// TwinCAT 3 PLC project Untitled1
// ProgramVersion: 3.1.4024.0
// libraries:
//   Tc2_MC2, * (Beckhoff Automation GmbH)
//   Tc2_SerialCom, * (Beckhoff Automation GmbH)
//   Tc2_Standard, * (Beckhoff Automation GmbH)
//   Tc2_System, * (Beckhoff Automation GmbH)
//   Tc3_Module, * (Beckhoff Automation GmbH)
// project tree:
//   DUTs/ tDataFrame.TcDUT
//   GVLs/ GVL.TcGVL
//   / PlcTask.TcTTO, RS485task.TcTTO
//   POUs/ FB_Azimuth.TcPOU, FB_Elevation.TcPOU, FB_485.TcPOU, FB_Trinamic_motors.TcPOU, MAIN.TcPOU, RS485_prg.TcPOU
// real-time tasks:
//   TASK PlcTask: cycle T#10ms, priority 20, ADS port 350
//   TASK RS485task: cycle T#1ms, priority 21, ADS port 352
// motion (NC):
//   TASK NC-Task 1 SAF: cycle T#2ms, priority 4, ADS port 501
//   TASK NC-Task 1 SVB: cycle T#10ms, priority 8, ADS port 511
//   AXIS Axis 3 (id 3)
//     General: UnitName=°
//     Dynamic: Acceleration=15000, Deceleration=15000, Jerk=64125
//     Velo: RefSearch=142.5, RefSync=142.5, SlowManual=712.5, FastManual=4275, Fast=14250, Maximum=14250
//     PositionAreaControl: Enable=false
//     TargetPosControl: Enable=false
//     OtherSettings: AllowMotionCmdToSlave=true
//     encoder EncType=8
//       EncPara: ScaleFactorNumerator=360, ScaleFactorDenominator=1048576, MaxCount=#xffffffff, EncPositionSource=1
//     drive DrvType=9
//       DrvPara: MaxCount=#xffffffff, DriveControlDWord=#x00030100
//         Analog: VeloReferenz=15675, VeloScale=1.02400649589962, TorqueSetpointScale=10, ScaleFactorActTorque=0.1
//         TimeComp: TaskDelayCycles=1
//     controller CtrType=1
//       CtrPara: PriorControlFactor=1
//         PosDiffControl: Enable=false
//         Observer: BandWidth=20
// I/O:
//   DEVICE Device 1 (EtherCAT), AmsNetId 5.79.241.154.2.1
//     Term 1 (EK1200) [EK1200-5000 EtherCAT Power supply (2A E-Bus)]
//       Term 2 (EL7342) [EL7342 2Ch. DC motor output stage (50V, 3.5A)]
//       RS485_term [EL6021 Interface (RS422/485)]
//       Term 3 (EK1110) [EK1110 EtherCAT extension]
//     Drive 4 (AX5203-0000-0214) [AX5203-0000-0214 EtherCAT Drive (SoE, 2 Ch.)]
// variable links:
//   NC-Task 1 SAF/Axes/Axis 3 <-> Device 1 (EtherCAT)/Drive 4 (AX5203-0000-0214)
//     Drive/Inputs/In/nDataIn1 <-> AT 1/Following distance
//     Drive/Inputs/In/nDataIn3[0] <-> AT 1/Torque/force feedback value
//     Drive/Inputs/In/nDcOutputTime <-> InfoData/DcOutputShift
//     Drive/Inputs/In/nState1 <-> AT 1/Drive status word @bit 8
//     Drive/Inputs/In/nState2 <-> AT 1/Drive status word
//     Drive/Inputs/In/nState4 @bit 1 <-> WcState/InputToggle
//     Drive/Inputs/In/nState4 <-> WcState/WcState
//     Drive/Outputs/Out/nCtrl1 <-> MDT 1/Master control word @bit 8
//     Drive/Outputs/Out/nDataOut1 <-> MDT 1/Position command value
//     Enc/Inputs/In/nDataIn1 <-> AT 1/Position feedback 1 value
//     Enc/Inputs/In/nDcInputTime <-> InfoData/DcInputShift
//     Enc/Inputs/In/nState4 @bit 1 <-> WcState/InputToggle
//     Enc/Inputs/In/nState4 <-> WcState/WcState
//   Untitled1/Untitled1 Instance <-> Device 1 (EtherCAT)/Term 1 (EK1200)/Term 2 (EL7342)
//     PlcTask Inputs/MAIN.Elevation.Encoder_Value <-> ENC Status Channel 1/Counter value
//     PlcTask Inputs/MAIN.Elevation.Error <-> DCM Status Channel 1/Status/Error
//     PlcTask Inputs/MAIN.Elevation.Homing_Switch <-> DCM Status Channel 1/Status/Digital input 1
//     PlcTask Inputs/MAIN.Elevation.Limit_Switch <-> DCM Status Channel 1/Status/Digital input 2
//     PlcTask Inputs/MAIN.Elevation.Moving_negative <-> DCM Status Channel 1/Status/Moving negative
//     PlcTask Inputs/MAIN.Elevation.Moving_positive <-> DCM Status Channel 1/Status/Moving positive
//     PlcTask Inputs/MAIN.Elevation.Ready <-> DCM Status Channel 1/Status/Ready
//     PlcTask Inputs/MAIN.Elevation.Warning <-> DCM Status Channel 1/Status/Warning
//     PlcTask Outputs/MAIN.Elevation.Enable <-> DCM Control Channel 1/Control/Enable
//     PlcTask Outputs/MAIN.Elevation.Encoder_Setvalue <-> ENC Control Channel 1/Set counter value
//     PlcTask Outputs/MAIN.Elevation.Reset <-> DCM Control Channel 1/Control/Reset
//     PlcTask Outputs/MAIN.Elevation.Set_Encoder <-> ENC Control Channel 1/Control/Set counter
//     PlcTask Outputs/MAIN.Elevation.Target_Position <-> DCM Position Channel 1/Position
//   Untitled1/Untitled1 Instance <-> NC-Task 1 SAF/Axes/Axis 3
//     PlcTask Inputs/MAIN.Azimuth.Azimuth_axis.NcToPlc <-> Outputs/ToPlc
//     PlcTask Outputs/MAIN.Azimuth.Azimuth_axis.PlcToNc <-> Inputs/FromPlc

CONFIGURATION Untitled1
    RESOURCE PLC ON TwinCAT3
        TASK PlcTask(INTERVAL := T#10ms, PRIORITY := 20);
        TASK RS485task(INTERVAL := T#1ms, PRIORITY := 21);
        PROGRAM MAIN WITH PlcTask : MAIN;
        PROGRAM RS485_prg WITH RS485task : RS485_prg;
    END_RESOURCE
END_CONFIGURATION

// ---- DUTs/tDataFrame.TcDUT
TYPE tDataFrame : ARRAY[0..8] OF BYTE; END_TYPE

// ---- GVLs/GVL.TcGVL
{attribute 'qualified_only'}
VAR_GLOBAL


nSetBaudrate : DINT := 38400;	
	
	
		{attribute 'TcLinkTo' := '
								.D[0]   := TIIB[RS485_term]^COM TxPDO-Map Inputs^Data In 0;
                              	.D[1]   := TIIB[RS485_term]^COM TxPDO-Map Inputs^Data In 1;
								.D[2]   := TIIB[RS485_term]^COM TxPDO-Map Inputs^Data In 2;
								.D[3]   := TIIB[RS485_term]^COM TxPDO-Map Inputs^Data In 3;
								.D[4]   := TIIB[RS485_term]^COM TxPDO-Map Inputs^Data In 4;
								.D[5]   := TIIB[RS485_term]^COM TxPDO-Map Inputs^Data In 5;
								.D[6]   := TIIB[RS485_term]^COM TxPDO-Map Inputs^Data In 6;
								.D[7]   := TIIB[RS485_term]^COM TxPDO-Map Inputs^Data In 7;
								.D[8]   := TIIB[RS485_term]^COM TxPDO-Map Inputs^Data In 8;
								.D[9]   := TIIB[RS485_term]^COM TxPDO-Map Inputs^Data In 9;
								.D[10]  := TIIB[RS485_term]^COM TxPDO-Map Inputs^Data In 10;
								.D[11]  := TIIB[RS485_term]^COM TxPDO-Map Inputs^Data In 11;
								.D[12]  := TIIB[RS485_term]^COM TxPDO-Map Inputs^Data In 12;
								.D[13]  := TIIB[RS485_term]^COM TxPDO-Map Inputs^Data In 13;
								.D[14]  := TIIB[RS485_term]^COM TxPDO-Map Inputs^Data In 14;
								.D[15]  := TIIB[RS485_term]^COM TxPDO-Map Inputs^Data In 15;
								.D[16]  := TIIB[RS485_term]^COM TxPDO-Map Inputs^Data In 16;
								.D[17]  := TIIB[RS485_term]^COM TxPDO-Map Inputs^Data In 17;
								.D[18]  := TIIB[RS485_term]^COM TxPDO-Map Inputs^Data In 18;
								.D[19]  := TIIB[RS485_term]^COM TxPDO-Map Inputs^Data In 19;
								.D[20]  := TIIB[RS485_term]^COM TxPDO-Map Inputs^Data In 20;
								.D[21]  := TIIB[RS485_term]^COM TxPDO-Map Inputs^Data In 21;
								.Status := TIIB[RS485_term]^COM TxPDO-Map Inputs^Status'}							  
	COMin_EL6021_MASTER AT %I* : EL6inData22B;              

			{attribute 'TcLinkTo' := '
								.D[0]   := TIIB[RS485_term]^COM RxPDO-Map Outputs^Data Out 0;
                              	.D[1]   := TIIB[RS485_term]^COM RxPDO-Map Outputs^Data Out 1;
								.D[2]   := TIIB[RS485_term]^COM RxPDO-Map Outputs^Data Out 2;
								.D[3]   := TIIB[RS485_term]^COM RxPDO-Map Outputs^Data Out 3;
								.D[4]   := TIIB[RS485_term]^COM RxPDO-Map Outputs^Data Out 4;
								.D[5]   := TIIB[RS485_term]^COM RxPDO-Map Outputs^Data Out 5;
								.D[6]   := TIIB[RS485_term]^COM RxPDO-Map Outputs^Data Out 6;
								.D[7]   := TIIB[RS485_term]^COM RxPDO-Map Outputs^Data Out 7;
								.D[8]   := TIIB[RS485_term]^COM RxPDO-Map Outputs^Data Out 8;
								.D[9]   := TIIB[RS485_term]^COM RxPDO-Map Outputs^Data Out 9;
								.D[10]  := TIIB[RS485_term]^COM RxPDO-Map Outputs^Data Out 10;
								.D[11]  := TIIB[RS485_term]^COM RxPDO-Map Outputs^Data Out 11;
								.D[12]  := TIIB[RS485_term]^COM RxPDO-Map Outputs^Data Out 12;
								.D[13]  := TIIB[RS485_term]^COM RxPDO-Map Outputs^Data Out 13;
								.D[14]  := TIIB[RS485_term]^COM RxPDO-Map Outputs^Data Out 14;
								.D[15]  := TIIB[RS485_term]^COM RxPDO-Map Outputs^Data Out 15;
								.D[16]  := TIIB[RS485_term]^COM RxPDO-Map Outputs^Data Out 16;
								.D[17]  := TIIB[RS485_term]^COM RxPDO-Map Outputs^Data Out 17;
								.D[18]  := TIIB[RS485_term]^COM RxPDO-Map Outputs^Data Out 18;
								.D[19]  := TIIB[RS485_term]^COM RxPDO-Map Outputs^Data Out 19;
								.D[20]  := TIIB[RS485_term]^COM RxPDO-Map Outputs^Data Out 20;
								.D[21]  := TIIB[RS485_term]^COM RxPDO-Map Outputs^Data Out 21;
								.Ctrl   := TIIB[RS485_term]^COM RxPDO-Map Outputs^Ctrl'}	
	COMout_EL6021_MASTER AT %Q* : EL6outData22B;
	RxBuffer_MASTER : Combuffer;
	TxBuffer_MASTER : Combuffer;	

END_VAR

// ---- POUs/MAIN.TcPOU
PROGRAM MAIN
VAR
Elevation : FB_Elevation;
Azimuth : FB_Azimuth;
END_VAR

Elevation();
Azimuth();

END_PROGRAM

// ---- POUs/FB_Elevation.TcPOU
FUNCTION_BLOCK FB_Elevation
VAR_INPUT
END_VAR
VAR_OUTPUT
END_VAR
VAR
	
	//Data for ADS communtication
	Targetpos_mm 			: LREAL	:= 0;		//Data FROM ADS
	Targetpos_deg			: LREAL := 0;		//Data FROM ADS
	Current_Position_mm 	: LREAL;			//Data TO ADS
	Current_Position_deg 	: LREAL; 			//Data from inclonometer, updated asynchronous from RS485
	Enable AT %Q* 			: BOOL 	:= FALSE;	//Data FROM ADS
	Homeing 				: BOOL 	:= FALSE;	//Data TO ADS
	Homeing_Error 			: BOOL 	:= FALSE;	//Data TO ADS
	Homeing_Wrong_direction : BOOL  := FALSE;	//Data TO ADS
	Reset_requested 		: BOOL  := FALSE;	//Data FROM ADS
	Error AT %I* 			: BOOL;				//Data TO ADS
	Target_in_deg			: BOOL  := FALSE;	//DATA FROM ADS
	//Position_Error AT %I* 	: BOOL;
	
		
	//Data for ADS communtication END
	
	
	Reset AT %Q* 			: BOOL 	:= FALSE;
	Encoder_Value AT %I* : UDINT;
	Homing_Switch AT %I* : BOOL;
	Limit_Switch AT %I* : BOOL;
	Warning AT %I* : BOOL;

	Ready AT %I* : BOOL;
	Moving_positive AT %I* : BOOL;
	Moving_negative AT %I* : BOOL;
	//In_target AT %I* : BOOL;
	Set_Encoder AT %Q* : BOOL;
	Encoder_Setvalue AT %Q* : UDINT;
	Target_Position AT %Q* : UDINT;
	
	P_error : LREAL; //position error
	Ang_P_fac : REAL := 0.01; //This is not really a P factor, I think it's more of a I
 	//Ang_I_fac : REAL := 0.001;

	
	//firstrun :BOOL := TRUE;
	Homed : BOOL := FALSE;
	Homeing_Allowed : BOOL := TRUE;
	Homeing_State : UINT := 0;
	Reset_state : UINT := 0;
	
	Homing_started_mm : LREAL; // to monitor if the homeing goes the right direction
	
	Homeing_Timer : TON; //used for timeouts
	Homeing_Timer2 : TON;
END_VAR

VAR CONSTANT
	maxmove_mm : LREAL := 210;
	minmove_mm : LREAL := 0;
	Zeroposition : UDINT := 1000000;
END_VAR

IF Homeing_Error THEN
	enable := FALSE;
	Homeing_state := 0;
	Homed := FALSE;
END_IF

IF Reset_requested THEN
	Reset_Elevation();
END_IF

IF Homed = FALSE AND Enable = TRUE AND Homeing_Allowed AND Homeing_Error = FALSE THEN
	//The homing sequence should start automaticly if the PLC is restarted and Enable is set
	Homeing_sequence();
ELSE
	IF Homed = TRUE AND Enable = TRUE THEN //Normal operation
		IF Target_in_deg = FALSE THEN
			//'Dumb' positioning, semi-openloop the position is only based on the 
			//Encoder value, not the actual measured value
			Target_Position := mm_to_encoder(LIMIT(minmove_mm,targetpos_mm,maxmove_mm));
		ELSE
			//closed-loop positionin with a inclonometer in the loop
			P_error := Current_Position_deg - Targetpos_deg;
			Target_Position := mm_to_encoder(LIMIT(minmove_mm,
			Target_Position + P_error*Ang_P_fac
			,maxmove_mm));
		END_IF
	
	
		
	END_IF
END_IF

current_position_mm := encoder_to_mm(Encoder_Value);

METHOD encoder_to_mm : LREAL
VAR_INPUT
	encoder_pos : UDINT;
END_VAR

VAR
	encoder_ppr : LREAL := 2000;
	mm_per_rev : LREAL := 0.8; //calibrate this value
END_VAR
encoder_to_mm := UDINT_TO_LREAL(encoder_pos - Zeroposition) / (encoder_ppr * mm_per_rev);
END_METHOD

METHOD Homeing_sequence : BOOL
VAR_INPUT
END_VAR
VAR
	diff_pos : LREAL;
END_VAR
Homeing_Timer(IN:=TRUE, PT:= T#200S); //timeout of the homeing, it takes a long time to home...
Homeing := TRUE;

IF Homeing_Timer.Q THEN
	//Timeout as been reached
	Homeing_Error := TRUE;
	Homeing_Timer(IN:=FALSE);

END_IF

IF Homing_Switch AND Homeing_state < 3 THEN
	Homeing_state := 3;
END_IF

CASE Homeing_state OF
	0:
	 	//We want to set the current position to a high number so we can go into the negative as the countervalue is a UDINT
		Encoder_Setvalue := Zeroposition;
		Target_Position  := Zeroposition;
		Set_Encoder := 1;
		Homeing_Timer2(IN:= TRUE, PT:= T#1S);
		IF Homeing_Timer2.Q THEN
			Homeing_Timer2(IN:=FALSE);
			Homeing_state := 1;
		END_IF
			
	1:
		Set_Encoder := 0;
		
		Homeing_Timer2(IN:= TRUE, PT:= T#1S);
		IF Homeing_Timer2.Q THEN
			Homeing_Timer2(IN:=FALSE);
			Homeing_state := 2;
			Homing_started_mm := encoder_to_mm(Encoder_Value);
		END_IF
	2: 
		//Goes to a position in the 'negatives' 
		Target_Position := 0;
		diff_pos := (encoder_to_mm(Encoder_Value) - Homing_started_mm);
		//Diff_pos will be very large if it is going the correct direction due to underflow
		//If it does not grow large, it is going the wrong way 
		IF  diff_pos > 1 AND diff_pos < 1000 THEN
			// for some reason this happens sometime
			homeing_error := TRUE;
			Homeing_Wrong_direction := TRUE;
		END_IF
		
	3: 
		//Stop the motor and set the new zero when the motor has stopped
		Target_Position := Encoder_Value; //Stop the motor without disabling it
		Homeing_Timer2(IN:= TRUE, PT:= T#2S);
		IF Homeing_Timer2.Q THEN
			Encoder_Setvalue := Zeroposition;
			Target_Position := Zeroposition;
			Set_Encoder := 1;
			Homeing_state := 4;
			Homeing_Timer2(IN:=FALSE);
		END_IF
		
	4: 
	
		//Motor has been homed
		Set_Encoder := 0;
		Homeing_Timer(IN:=FALSE);
		Homeing := FALSE;
		Homed := TRUE;
		homeing_state := 0;
		
	
END_CASE
END_METHOD

METHOD mm_to_encoder : UDINT
VAR_INPUT
	mm_in : LREAL;
END_VAR
VAR
	encoder_ppr : LREAL := 2000;
	mm_per_rev : LREAL := 0.8; //calibrate this value
END_VAR
mm_to_encoder := LREAL_TO_UDINT(mm_in* mm_per_rev * encoder_ppr) + Zeroposition;
END_METHOD

METHOD Reset_Elevation : BOOL
VAR_INPUT
END_VAR

CASE Reset_state OF
	0:
		enable := FALSE;
		Reset_state := 1;
	1:
		Reset := TRUE;
		Targetpos_mm := Current_Position_mm ;
		Homed := FALSE;
		Homeing_Error := FALSE;
		Homeing_Wrong_direction := FALSE;
		Homeing_State := 0;
		Reset_state := 2;
		
	2: 
		Reset := FALSE;
		Reset_state := 3;
		
	3: //A extra one for good luck
		Reset := TRUE;
		Reset_state := 3;
		
	4: 
		Reset := FALSE;
		Reset_state := 0;
		Reset_requested := FALSE;
	
END_CASE
END_METHOD

METHOD set_Current_Position_deg : BOOL
VAR_INPUT
	deg : LREAL;
END_VAR
Current_Position_deg := deg;
END_METHOD

END_FUNCTION_BLOCK

// ---- POUs/FB_Azimuth.TcPOU
FUNCTION_BLOCK FB_Azimuth
VAR
	
	EnableAzimuth : BOOL := FALSE; //For ADS


	Azimuth_Target_Position_Parabola : LREAL := 0; // for ADS, target position in 'real' angles
	HMI_Azimuth : LREAL; //Readable position, scaled for your pleasure for ADS
	
	Azimuth_target_position : LREAL := 0; //in motor angles, 
	
	Azimuth_CurrentPosition : LREAL;
	Azimuth_Old_position : LREAL;
	Azimuth_Moveto_position :LREAL;
	Azimuth_state : INT := 1;
	Azimuth_enable_tracking : BOOL := FALSE;
	Azimuth_setpoint_scaled: REAL;
	Azimuth_actual_position : LREAL;
	
	Azimuth_axis : AXIS_REF; 
	Azimuth_PowerAxis: MC_Power;
	Azimuth_PowerAxisOut: ST_McOutputs;
	Azimuth_MoveAxis: MC_MoveAbsolute;
	Azimuth_MoveAbsoluteOut: ST_McOutputs;
	Azimuth_ResetOut: ST_McOutputs;
	

	Azimuth_Axis_power : MC_Power;
	Azimuth_axis_move_abs : MC_moveAbsolute;
	Azimuth_Reset : MC_Reset;
	
	Azimuth_timer : TON; //Timer for init of Azimuth_axis
END_VAR

VAR CONSTANT
	Azimuth_zero : REAL := 0; //'fake' zero position
	Gearratio : REAL := 0.0011904761904762;//1.0/840.0;

END_VAR


IF EnableAzimuth = FALSE THEN
	Azimuth_state := 0;
END_IF

IF EnableAzimuth = TRUE AND Azimuth_state = 0 THEN
	Azimuth_state := 1;
END_IF
 
 update_Azimuth();

METHOD update_Azimuth : BOOL
VAR_INPUT
END_VAR
VAR CONSTANT
	Invert_Azimuth_axis : BOOL := FALSE;
END_VAR
Azimuth_axis();

Azimuth_target_position := Azimuth_Target_Position_Parabola/gearratio;

IF Invert_Azimuth_axis THEN
	Azimuth_setpoint_scaled := Azimuth_target_position;
	Azimuth_CurrentPosition := Azimuth_axis.NcToPlc.ActPos;
	Azimuth_actual_position := Azimuth_axis.NcToPlc.ActPos - Azimuth_zero;
	
	Azimuth_Moveto_position := Azimuth_zero + Azimuth_target_position; 
ELSE
	Azimuth_setpoint_scaled := Azimuth_target_position;
	Azimuth_CurrentPosition := Azimuth_axis.NcToPlc.ActPos;
	Azimuth_actual_position := Azimuth_zero - Azimuth_axis.NcToPlc.ActPos;
	
	Azimuth_Moveto_position := Azimuth_zero - Azimuth_target_position; 

END_IF
CASE Azimuth_state OF
	-1 : //Error state
			IF Azimuth_axis.Status.Error THEN
				Azimuth_state := 4;	(* axis error requires reset *)
			ELSE
				Azimuth_state := 1;	(* function block errors don't need a reset *)
			END_IF
		
	0 : //Stopped
			Azimuth_MoveAxis.Execute := FALSE;
			Azimuth_PowerAxis.Enable := FALSE;
			Azimuth_PowerAxis.Enable_Positive := FALSE;
			Azimuth_PowerAxis.Enable_Negative := FALSE;
	1 : //INIT
			Azimuth_MoveAxis.Execute := FALSE;
			Azimuth_Reset.Execute := FALSE;
			Azimuth_state := 2;	
			IF Azimuth_PowerAxis.Error THEN
				Azimuth_state := -1;
			END_IF
	2 : //Enabled but not moving
			Azimuth_PowerAxis.Enable := TRUE;
			Azimuth_PowerAxis.Enable_Positive := TRUE;
			Azimuth_PowerAxis.Enable_Negative := TRUE;
			Azimuth_MoveAxis.BufferMode := MC_aborting;
			IF EnableAzimuth AND Azimuth_axis.Status.Operational THEN
				Azimuth_state := 33;
				Azimuth_enable_tracking := TRUE;
			END_IF
			
			IF Azimuth_PowerAxis.Error THEN
				Azimuth_state := -1;
			END_IF
	
	33 : //Tracking mode, tries to follow Azimuth value 

		
			//Pulse .Execute since movement is triggered on rising edge
			IF Azimuth_MoveAxis.Execute THEN
				Azimuth_MoveAxis.Execute := FALSE;
			ELSE
				//IF movements are large enough
				IF ABS(Azimuth_Moveto_position - Azimuth_axis.NcToPlc.ActPos) > 0.04 OR ABS(Azimuth_Moveto_position - Azimuth_Old_position) > 0.04 THEN
					Azimuth_Old_position := Azimuth_Moveto_position;
					Azimuth_MoveAxis.Position := Azimuth_Moveto_position;
					Azimuth_MoveAxis.Acceleration  := 40_000;
					Azimuth_MoveAxis.Deceleration  := 40_000;
					Azimuth_MoveAxis.Jerk 			:= 10_000;
					Azimuth_MoveAxis.Velocity 		:= 14000;

					Azimuth_MoveAxis.Execute 		:= TRUE;
					
				ELSE
					Azimuth_MoveAxis.Execute := FALSE;
				END_IF
			END_IF

			IF Azimuth_enable_tracking = FALSE THEN //If tracking is no longer desired
				Azimuth_state := 2;
			END_IF
			IF Azimuth_MoveAxis.CommandAborted OR Azimuth_MoveAxis.Error OR Azimuth_axis.Status.Error THEN //Machine error
				Azimuth_state := -1;
			END_IF
			
	4: //Reset
			Azimuth_Reset.Execute := TRUE;
			IF Azimuth_Reset.Done THEN
				Azimuth_state := 1;
			ELSIF Azimuth_Reset.Error THEN
				Azimuth_state := 1; 
			END_IF

END_CASE


IF Invert_Azimuth_axis THEN
	HMI_Azimuth := Azimuth_axis.NcToPlc.ActPos*gearratio - Azimuth_zero;
ELSE
	HMI_Azimuth := Azimuth_zero - Azimuth_axis.NcToPlc.ActPos*gearratio;

END_IF

Azimuth_Axis_power(		
	Axis:=Azimuth_axis,
	Enable:=Azimuth_PowerAxis.Enable,
	Enable_positive:=Azimuth_PowerAxis.Enable_Positive,
	Enable_negative:=Azimuth_PowerAxis.Enable_Negative,
	Override:=100,
	Status =>Azimuth_PowerAxisOut.done,
	Busy=>Azimuth_PowerAxisOut.Busy,
	Active=>Azimuth_PowerAxisOut.Active,
	Error=>Azimuth_PowerAxisOut.Error,
	ErrorID => Azimuth_PowerAxisOut.ErrorID
);

Azimuth_axis_move_abs(
	Axis:=Azimuth_axis,
	execute:=Azimuth_MoveAxis.Execute,
	Position:=Azimuth_MoveAxis.Position,
	Velocity:=Azimuth_MoveAxis.Velocity,
	Acceleration:=Azimuth_MoveAxis.Acceleration,
	Deceleration:=Azimuth_MoveAxis.Deceleration,
	BufferMode:=Azimuth_MoveAxis.BufferMode,
	Jerk:=Azimuth_MoveAxis.Jerk,
	Done=>Azimuth_MoveAbsoluteOut.Done,
	Busy=>Azimuth_MoveAbsoluteOut.Busy,
	Active=>Azimuth_MoveAbsoluteOut.Active,
	CommandAborted=>Azimuth_MoveAbsoluteOut.CommandAborted,
	Error=>Azimuth_MoveAbsoluteOut.Error,
	ErrorID=>Azimuth_MoveAbsoluteOut.ErrorID
);

Azimuth_Reset(
	Axis:=Azimuth_axis,
	Execute:=Azimuth_Reset.Execute,
	Busy=>Azimuth_ResetOut.Busy,
	Error=>Azimuth_ResetOut.Error,
	ErrorID=>Azimuth_ResetOut.ErrorID
);
END_METHOD

END_FUNCTION_BLOCK

// ---- POUs/RS485_prg.TcPOU
PROGRAM RS485_prg
VAR
	
	COMportControl_MASTER: SerialLineControl;
	COMportControlError_MASTER : BOOL;
	COMportControlErrorID_MASTER : ComError_t;	

END_VAR



COMportControl_MASTER(
	Mode:=SERIALLINEMODE_EL6_22B,
	pComIn:= ADR(GVL.COMin_EL6021_MASTER),
	pComOut:= ADR(GVL.COMout_EL6021_MASTER),
	SizeComIn:= UINT_TO_INT(SIZEOF(GVL.COMin_EL6021_MASTER)),
	TxBuffer:= GVL.TxBuffer_MASTER,
	RxBuffer:=GVL.RxBuffer_MASTER,
	Error => COMportControlError_MASTER,
	ErrorID => COMportControlErrorID_MASTER);

END_PROGRAM

// ---- POUs/FB_485.TcPOU
FUNCTION_BLOCK FB_485
//This functionblock is suposed to handle the 485 comminication
VAR_INPUT
END_VAR
VAR_OUTPUT
END_VAR
VAR
	
	Timer : TON;
	//timer2 : TON;
	Send: SendData; //Functionblock of TC2_SerialCom
	SendBusy: BOOL; // copy of SendData.Busy
	SendErrorID: ComError_t;
	aDataTx: tDataFrame;
	Receive: ReceiveData;
	LastReceivedDataBytes: tDataFrame;
	DataReceived: BOOL;
	ReceiveBusy: BOOL;
	ReceiveErrorID: ComError_t;
	ReceiveTimeout: BOOL;
	ReceiveCounter: UDINT :=0;	
	aDataRx: tDataFrame;
	nDataLen: BYTE := 9;
	bNodeId_SL1: BYTE := 1; //Slave one Serial ID
	nState: INT;
	nRxChecksum: BYTE;
	nCalcChecksum: BYTE;
	T_ReceiveDelay:TIME;
	
	//Used as a intermediate step to transmit/recive
	RXcombuffer : combuffer;
	TXcombuffer : combuffer;
	Combuffersize : UINT := 301;//0..300 so 301 values //Defined by combuffer
	
	RegisterRequested : BOOL := FALSE;
	AxisParameterRequested : BOOL := FALSE;

	i: UINT;
END_VAR
VAR CONSTANT
	
END_VAR

METHOD DataRequestHandler : BOOL
VAR_INPUT
END_VAR
VAR
	payload : DWORD;
	Module : BYTE;
	Fcode : BYTE;
	msg_len : BYTE;
	Command : BYTE;
	i : BYTE;
	Checksum: UINT;
	Checksum_rec : UINT;
	REQ_data : ARRAY[0 .. 8] OF BYTE;
	last_issued_get_index : UINT;
END_VAR
IF RXcombuffer.Count > 1 THEN
	
	//This is done instead of a memcpy as RXcombuffer is a ringbuffer and the loopover is scary
	//Debug data mainly
	REQ_data[0] := RXcombuffer.Buffer[(RXcombuffer.RdIdx+0) MOD Combuffersize];
	REQ_data[1] := RXcombuffer.Buffer[(RXcombuffer.RdIdx+1) MOD Combuffersize];
	REQ_data[2] := RXcombuffer.Buffer[(RXcombuffer.RdIdx+2) MOD Combuffersize];
	REQ_data[3] := RXcombuffer.Buffer[(RXcombuffer.RdIdx+3) MOD Combuffersize];
	REQ_data[4] := RXcombuffer.Buffer[(RXcombuffer.RdIdx+4) MOD Combuffersize];
	REQ_data[5] := RXcombuffer.Buffer[(RXcombuffer.RdIdx+5) MOD Combuffersize];
	REQ_data[6] := RXcombuffer.Buffer[(RXcombuffer.RdIdx+6) MOD Combuffersize];
	REQ_data[7] := RXcombuffer.Buffer[(RXcombuffer.RdIdx+7) MOD Combuffersize];
	REQ_data[8] := RXcombuffer.Buffer[(RXcombuffer.RdIdx+8) MOD Combuffersize];
	REQ_data[9] := RXcombuffer.Buffer[(RXcombuffer.RdIdx+9) MOD Combuffersize];
	REQ_data[10] := RXcombuffer.Buffer[(RXcombuffer.RdIdx+10) MOD Combuffersize];
	REQ_data[11] := RXcombuffer.Buffer[(RXcombuffer.RdIdx+11) MOD Combuffersize];
	REQ_data[12] := RXcombuffer.Buffer[(RXcombuffer.RdIdx+12) MOD Combuffersize];
	REQ_data[13] := RXcombuffer.Buffer[(RXcombuffer.RdIdx+13) MOD Combuffersize];
	
//	last_issued_get_index := (TXcombuffer.WrIdx-6 MOD Combuffersize); //Should uilize aTX buffer instead
	
	Module  := RXcombuffer.Buffer[(RXcombuffer.RdIdx+1) MOD Combuffersize]; //Adress
	Fcode  := RXcombuffer.Buffer[(RXcombuffer.RdIdx+2) MOD Combuffersize]; // Function code
	msg_len := RXcombuffer.Buffer[(RXcombuffer.RdIdx+3) MOD Combuffersize]; //Byte length, of data, not including CRC and header
	
	//Cecksum is 16-bit, combine two bytes( 4+msg_len )
	Checksum_rec := payload := (RXcombuffer.Buffer[RXcombuffer.RdIdx+( 5+msg_len ) MOD Combuffersize] 
	OR SHR(BYTE_TO_DWORD(RXcombuffer.Buffer[(RXcombuffer.RdIdx+( 4+msg_len )) MOD Combuffersize]),8));
	
	//Checksum := RXcombuffer.Buffer[(RXcombuffer.RdIdx) MOD Combuffersize];
	//FOR i := 1 TO 7 DO
	//	Checksum := Checksum + RXcombuffer.Buffer[(RXcombuffer.RdIdx+i) MOD Combuffersize];
	//END_FOR
	
	//IF Checksum = Checksum_rec THEN
		//If the checksum is correct
	
		CASE Fcode OF

			3: //Return data of angle
			IF RegisterRequested THEN
				RegisterRequested := FALSE;
				payload := (RXcombuffer.Buffer[RXcombuffer.RdIdx+7 MOD Combuffersize] 
				OR SHR(BYTE_TO_DWORD(RXcombuffer.Buffer[(RXcombuffer.RdIdx+6) MOD Combuffersize]),8) 
				OR SHR(BYTE_TO_DWORD(RXcombuffer.Buffer[(RXcombuffer.RdIdx+5) MOD Combuffersize]),16) 
				OR SHR(BYTE_TO_DWORD(RXcombuffer.Buffer[(RXcombuffer.RdIdx+4) MOD Combuffersize]),24));

			END_IF
			
		END_CASE
	//ELSE
	//	//Invalid checksum
	//	ADSLOGSTR(msgCtrlMask:=ADSLOG_MSGTYPE_ERROR,msgFmtStr:='Got an invalid RS485 checksum in DataRequestHandler',strArg:='');
	//END_IF
	
	RXcombuffer.Count := RXcombuffer.Count - nDataLen;
	RXcombuffer.RdIdx := ((RXcombuffer.RdIdx + nDataLen)  MOD Combuffersize);
	RXcombuffer.FreeByte := RXcombuffer.FreeByte + nDataLen;
END_IF
END_METHOD

METHOD fb_init : BOOL
VAR_INPUT
	bInitRetains : BOOL;
	bInCopyCode : BOOL;
END_VAR

VAR
	i: BYTE;
END_VAR
//PD1140 : ARRAY[1..3] OF TMCL_Motor;

FOR i := 1 TO nMotors DO
	PD1140[i].MotorID := i;
	RequestedPos[i] := 0;
END_FOR
PD1140[1].Offset := 0;
PD1140[2].Offset := 0;
PD1140[3].Offset := PD1140[2].Offset;
END_METHOD

METHOD RequestAxisParameter : BOOL
VAR_INPUT
	MotorID : BYTE;
	InstType : BYTE;
	Bank : BYTE;
END_VAR
VAR
	aDataTx: tDataFrame;
END_VAR
IF GVL.TxBuffer_MASTER.Count < 1 THEN //No other commands in the buffer, so add this
							//This is done to maintain priority for the wirefeed stuff and try to remove artifacts from reading

	AxisParameterRequested := TRUE; // This ties in with the DataRequestHandler
	aDataTX[0] := MotorID;
	aDataTX[1] := 6; 
	aDataTX[2] := InstType;
	aDataTX[3] := Bank;
	//DATA
	
	aDataTX[7] := 0;
	aDataTX[6] := 0;
	aDataTX[5] := 0;
	aDataTX[4] := 0;
	
	aDataTX[8] := 0; //Checksum is calcuated on transmit
	Transmit(dataIn := aDataTX);
	RequestAxisParameter := TRUE;
ELSE
	//The buffer has something in it, and nothing was sent
 	RequestAxisParameter := FALSE;
END_IF
END_METHOD

METHOD SendCycle : BOOL
VAR_INPUT
END_VAR

VAR

	i: UINT;
	
	Checksum: WORD;
	Trans_delay : TIME := LREAL_TO_TIME(nDataLen * (1/DINT_TO_LREAL(nSetBaudrate))*33*1000);
END_VAR
CASE nState OF
0:

timer(IN:=TRUE,PT:=Trans_delay);
IF Timer.Q THEN
	IF TXcombuffer.Count > 1 THEN
		
		//Extract a datapackage from the ringbuffer	
		IF TXcombuffer.RdIdx + nDataLen >= Combuffersize THEN
			//If the buffer loops around the edge
			FOR i := 0 TO nDataLen-1 DO
				aDataTX[i] := TXcombuffer.buffer[((TXcombuffer.RdIdx + i) MOD Combuffersize)];

			END_FOR
			TXcombuffer.Count := TXcombuffer.Count - nDataLen;
			TXcombuffer.FreeByte := TXcombuffer.FreeByte + nDataLen;
			TXcombuffer.RdIdx := ((TXcombuffer.RdIdx + nDataLen ) MOD Combuffersize);
		ELSE
			//Normal operation of the buffer
			memcpy(destAddr:=ADR(aDataTX), srcAddr:=ADR(TXcombuffer.buffer[TXcombuffer.RdIdx]) , nDataLen);
			TXcombuffer.Count := TXcombuffer.Count - nDataLen;
			TXcombuffer.RdIdx := ((TXcombuffer.RdIdx + nDataLen ) MOD Combuffersize);
			TXcombuffer.FreeByte := TXcombuffer.FreeByte + nDataLen;
		END_IF
		
		
		//Calculate checksum
		Checksum := aDataTX[0];
		FOR i := 1 TO 7 DO
			Checksum := Checksum + aDataTX[i];
		END_FOR
		//Checksum := Checksum MOD 255; //Potential unnecicary row
		aDataTX[8] := WORD_TO_BYTE(Checksum); //Overwrites the inputted checksum
		
		Send(pSendData:=ADR(aDataTX),Length :=nDataLen,
			TXbuffer:=TxBuffer_MASTER,
			Busy =>SendBusy, Error => SendErrorID);
		Timer(IN:=FALSE);
		IF NOT SendBusy THEN
			nState := nState+1;
		END_IF
	END_IF
END_IF

1:

	//T_ReceiveDelay := nDataLen *REAL_TO_TIME((1/DINT_TO_REAL(nSetBaudrate))*33*1000);
	timer(IN:=TRUE,PT:=Trans_delay);
	IF Timer.Q THEN
		nState:= nState+1;
		Timer(IN:=FALSE);
	END_IF
	
2:

Receive(
pReceiveData :=ADR(aDataRX[0]),
SizeReceiveData:= (nDataLen),
RXbuffer:= RxBuffer_MASTER,
Timeout:=T#1S,
DataReceived=>DataReceived,
busy => receiveBusy,
Error => ReceiveErrorID,
RxTimeout =>ReceiveTimeout);

IF DataReceived THEN
	IF NOT ReceiveBusy THEN
		nRxChecksum := aDataRX[nDataLen-1];
		
		Checksum := aDataRX[0];
		FOR i := 1 TO nDataLen-2 DO
			Checksum := Checksum + aDataRX[i];
		END_FOR
		//Checksum := Checksum MOD 255; //Potential unnecicary row
		nCalcChecksum := WORD_TO_BYTE(Checksum); //Overwrites the inputted checksum
		
		IF(nRXChecksum = nCalcChecksum) THEN
			IF RXcombuffer.WrIdx + nDataLen >= Combuffersize THEN
				//Loop around write
				FOR i := 0 TO nDataLen-1 DO
					RXcombuffer.buffer[((RXcombuffer.WrIdx + i) MOD Combuffersize)] := aDataRX[i];
				END_FOR
				RXcombuffer.Count := RXcombuffer.Count + nDataLen;
				RXcombuffer.FreeByte := RXcombuffer.FreeByte - nDataLen;
				RXcombuffer.WrIdx := ((RXcombuffer.WrIdx + nDataLen) MOD Combuffersize);
				
			ELSE	
				//Normal operation of the buffer
				memcpy( destAddr:=ADR(RXcombuffer.buffer[RXcombuffer.WrIdx]) , srcAddr:=ADR(aDataRX) , nDataLen);
				RXcombuffer.WrIdx := ((RXcombuffer.WrIdx + nDataLen) MOD Combuffersize);
				RXcombuffer.Count := RXcombuffer.Count + nDataLen;
				RXcombuffer.FreeByte := TXcombuffer.FreeByte - nDataLen;
			END_IF
		END_IF
		nState := 0;
	END_IF
	ELSE
		Timer(IN:=TRUE,PT:=T#50MS);
		IF Timer.Q THEN //Timeout
			nState := 0;
			RXcombuffer.WrIdx := ((RXcombuffer.WrIdx + nDataLen) MOD Combuffersize);
			RXcombuffer.FreeByte := TXcombuffer.FreeByte - nDataLen;
			RXcombuffer.Count := RXcombuffer.Count + nDataLen;
		END_IF
	END_IF
END_CASE
END_METHOD

METHOD SetAxisParameter : BOOL
VAR_INPUT
	MotorID : BYTE;
	InstType : BYTE;
	Bank : BYTE;
	data : DINT;
END_VAR
VAR
	aDataTx: tDataFrame;
END_VAR

aDataTX[0] := MotorID;
aDataTX[1] := 5; //SAP set axis parameter 
aDataTX[2] := InstType;
aDataTX[3] := Bank;
//DATA

aDataTX[7] := DINT_TO_BYTE(data);
data := SHR(data,8);
aDataTX[6] := DINT_TO_BYTE(data);
data := SHR(data,8);
aDataTX[5] := DINT_TO_BYTE(data);
data := SHR(data,8);
aDataTX[4] := DINT_TO_BYTE(data);

aDataTX[8] := 0; //Checksum is calcuated on transmit
Transmit(dataIn := aDataTX);
END_METHOD

METHOD Transmit : INT
VAR_INPUT
	dataIn : tDataFrame;
END_VAR

VAR
	i: UINT;
END_VAR
//Add data to the end of the transmit buffer
IF TXcombuffer.Count >= Combuffersize - nDataLen THEN
	TXcombuffer.Error := INT_TO_UINT(ComError_t.COMERROR_TXBUFFOVERRUN);
	Transmit := ComError_t.COMERROR_TXBUFFOVERRUN;
ELSE
	Transmit := ComError_t.COMERROR_NOERROR;
	TXcombuffer.Error := INT_TO_UINT(ComError_t.COMERROR_NOERROR);
	
	IF TXcombuffer.WrIdx + nDataLen >= Combuffersize THEN
		//Loop around write
		FOR i := 0 TO nDataLen-1 DO
			TXcombuffer.buffer[((TXcombuffer.WrIdx + i) MOD Combuffersize)] := dataIn[i];
		END_FOR
		TXcombuffer.WrIdx := ((TXcombuffer.WrIdx + nDataLen) MOD Combuffersize);
		TXcombuffer.Count := TXcombuffer.Count + nDataLen;
		TXcombuffer.FreeByte := TXcombuffer.FreeByte - nDataLen;
				
	ELSE	
		//Normal operation of the buffer
		memcpy( destAddr:=ADR(TXcombuffer.buffer[TXcombuffer.WrIdx]) , srcAddr:=ADR(dataIn) , nDataLen);
		TXcombuffer.Count := TXcombuffer.Count + nDataLen;
		TXcombuffer.WrIdx := ((TXcombuffer.WrIdx + nDataLen) MOD Combuffersize);
		TXcombuffer.FreeByte := TXcombuffer.FreeByte - nDataLen;
	END_IF
END_IF
END_METHOD

METHOD update : BOOL
VAR_INPUT
END_VAR
VAR

END_VAR
SendCycle();
DataRequestHandler();
//X := LREAL_TO_REAL(PD1140[1].GetPosition()*gearing-PD1140[1].Offset);
//Y := LREAL_TO_REAL(PD1140[2].GetPosition()*gearing-PD1140[2].Offset);
//Z := LREAL_TO_REAL(PD1140[3].GetPosition()*gearing-PD1140[3].Offset);
//
//X_temp := PD1140[1].Temperature;
//Y_temp := PD1140[2].Temperature;
//Z_temp := PD1140[3].Temperature;
WF_temp := PD1140[4].Temperature;
WF_current := PD1140[4].CurrentDraw;
END_METHOD

METHOD Update_TMCL_wirefeeder : BOOL
VAR_INPUT

END_VAR

VAR CONSTANT
	ID: BYTE := 4; //ID of the wiremotor
	
	Wheel_diameter : REAL := 22.45; //Adjusted after measuring a meter 22.79; // diameter of the feedwheel in mm //Outside diameter is 23.0, groove bottom is 22.7
	wire_diameter : REAL := 0.8; // in mm, Only used to calculate mass-flow
	gearing : LREAL := 12.5;//6.25;//12.5; // 12.5 rotations on the axle gives one roation of the wheel
END_VAR


VAR
	Setpoint_RPM : LREAL := 0;
	
	Dir : BOOL;
	SpeedError : BOOL := FALSE;
END_VAR
//Calculate the speed of the motor from feedrate
SpeedError := FALSE;
_Speed := 0;
IF(WireFeedrate > 0) THEN
	Dir := TRUE;
ELSIF(WireFeedrate <0) THEN
	DIR:= FALSE;
END_IF

//Feedrates uint is [mm/s]
Setpoint_RPM := ((ABS(WireFeedrate) * 60 * gearing) / (Wheel_diameter*3.1415));
_Speed := PD1140[4].CONVERT_RPM_TO_INTSPEED(Setpoint_RPM);


IF(_Speed > 2047) THEN
	_speed := 2047;
	SpeedError := TRUE;
ELSIF(_Speed < 0) THEN
	_Speed := 0;
	SpeedError := TRUE;
END_IF


IF (NOT (PD1140[ID].GetSpeed() = _Speed)) THEN //If a speedchange is neccesarry
	
	//Declare the direction of rotoation
	IF   (_Speed > 0) THEN
		RotateMotor(Speed := _Speed, MotorID := ID,Direction := Dir);
	ELSIF(_Speed = 0) THEN
		StopMotor(ID);
	END_IF
	PD1140[ID].SetSpeed(_Speed);

END_IF
END_METHOD

END_FUNCTION_BLOCK

// ---- POUs/FB_Trinamic_motors.TcPOU
FUNCTION_BLOCK FB_Trinamic_motors
VAR_INPUT
END_VAR
VAR_OUTPUT
END_VAR

VAR
	eDataReq : eReqestType;
	Trans_Timer : TON;
	//timer2 : TON;
	Send: SendData; //Functionblock of TC2_SerialCom
	BusBusy : BOOL;
	SendBusy: BOOL; // copy of SendData.Busy
	SendErrorID: ComError_t;
	aDataTx: tDataFrame;
	Receive: ReceiveData;
	LastReceivedDataBytes: tDataFrame;
	DataReceived: BOOL;
	ReceiveBusy: BOOL;
	ReceiveErrorID: ComError_t;
	ReceiveTimeout: BOOL;
	ReceiveCounter: UDINT :=0;	
	aDataRx: tDataFrame;
	nDataLen: BYTE := 9;
	bNodeId_SL1: BYTE := 1; //Slave one Serial ID

	nRxChecksum: BYTE;
	nCalcChecksum: BYTE;
	T_ReceiveDelay:TIME;

	 motors : ARRAY[1..4] OF TMCL_Motor; //IF YOU CAHNGE THIS CHANGE REQUESTHANDLER
	
END_VAR

METHOD FB_init : BOOL
VAR_INPUT
	bInitRetains : BOOL; // if TRUE, the retain variables are initialized (warm start / cold start)
	bInCopyCode : BOOL;  // if TRUE, the instance afterwards gets moved into the copy code (online change)
END_VAR

VAR
	i: UINT;
END_VAR
FOR i := 1 TO 3 DO
	motors[i].MotorID := UINT_TO_BYTE(i);
END_FOR
END_METHOD

METHOD Transmit : BYTE
VAR_INPUT
	Input : tDataFrame;
END_VAR
VAR
	Checksum : WORD;
	i: INT;
	//SendBusy : BOOL;
	//SendErrorID : ComError_t;
END_VAR

//Calculate Checksum NOTE byte 9 (checksum byte) is disregarded
Checksum := Input[0];
FOR i := 1 TO 7 DO
	Checksum := Checksum + Input[i];
END_FOR

Checksum := Checksum MOD 255; //Potential unnecicary row

Input[8] := WORD_TO_BYTE(Checksum); //Overwrites the inputted checksum

Send(pSendData:=ADR(Input),Length := 9,
		TXbuffer:=TxBuffer_MASTER,
		Busy =>SendBusy, Error => SendErrorID);

T_ReceiveDelay := REAL_TO_TIME((1/DINT_TO_REAL(nSetBaudrate))*33*1000);
Trans_timer(IN:=TRUE,PT:=T_ReceiveDelay);

BusBusy := TRUE;

Transmit := WORD_TO_BYTE(Checksum);
END_METHOD

METHOD Update : BOOL
VAR_INPUT
END_VAR
VAR
	Timer : TON;
	Checksum: WORD;
	i: INT;
END_VAR


IF Trans_timer.Q THEN
	Trans_timer(IN:=FALSE);
	Receive(
		pReceiveData := ADR(aDataRX),
		SizeReceiveData := (9),
		RXbuffer := RxBuffer_MASTER,
		Timeout:=T#1S,
		DataReceived=>DataReceived,
		busy => receiveBusy,
		Error => ReceiveErrorID,
		RxTimeout =>ReceiveTimeout);

		
	IF DataReceived THEN
		//ReceiveCounter := ReceiveCounter+1;
		IF NOT ReceiveBusy THEN
			
			//Calculate Checksum
			Checksum := aDataRX[0];
			FOR i := 1 TO 7 DO
				Checksum := Checksum + aDataRX[i];
			END_FOR
			
			//Only apply recived Data if the checksum is correct
			IF(aDataRX[8] = WORD_TO_BYTE(Checksum)) THEN
				memset(ADR(LastReceivedDataBytes[0]),0,(SIZEOF(aDataRX)-1));
				memcpy(ADR(LastReceivedDataBytes[0]),ADR(aDataRX),(nDataLen+1));
			END_IF
			BusBusy := FALSE;
		END_IF
		
	ELSE
		Timer(IN:=TRUE,PT:=T#0.1S);
		IF Timer.Q THEN //Timeout
			BusBusy := FALSE;
			eDataReq := eReqestType.NOREQ;
		END_IF	
	END_IF
	DataRequestHandler();
END_IF
END_METHOD

END_FUNCTION_BLOCK
